// Mitsubishi GX Works2 project: DGPTapM6FX3G   PLC: FX3G

// global labels: Global1
VAR_GLOBAL
  VR1 AT D8030 : INT;
  VR2 AT D8031 : INT;
  XXLimitN AT M8344 : BOOL;
  XXLimitP AT M8343 : BOOL;
  XXBusy AT M8340 : BOOL;
  XXInterruptInverse AT M8347 : BOOL;
  XXPos AT D8340 : DINT;
  XXAccelTime AT D8348 : INT;
  XXDecelTime AT D8349 : INT;
  XXPosView AT D0 : DINT;
  XXTarPos AT D2 : DINT;
  XXFeed AT D4 : DINT;
  XXTarR AT M0 : BOOL;
  XXTarRSkip AT D6 : INT;
  XXOn AT M1 : BOOL;
  XXRun AT M2 : BOOL;
  XXDirection AT M3 : BOOL;
  XXMinI AT X000 : BOOL;
  XXReadyI AT X003 : BOOL;
  XXPulseO AT Y000 : BOOL;
  XXDirectionO AT Y004 : BOOL;
  XXOnO AT Y002 : BOOL;
  YYLimitN AT M8354 : BOOL;
  YYLimitP AT M8353 : BOOL;
  YYBusy AT M8350 : BOOL;
  YYInterruptInverse AT M8357 : BOOL;
  YYPos AT D8350 : DINT;
  YYAccelTime AT D8358 : INT;
  YYDecelTime AT D8359 : INT;
  YYPosView AT D7 : DINT;
  YYTarPos AT D9 : DINT;
  YYFeed AT D11 : DINT;
  YYTarR AT M4 : BOOL;
  YYTarRSkip AT D13 : INT;
  YYOn AT M5 : BOOL;
  YYRun AT M6 : BOOL;
  YYDirection AT M7 : BOOL;
  YYMinI AT X001 : BOOL;
  YYMaxI AT X002 : BOOL;
  YYReadyI AT X004 : BOOL;
  YYPulseO AT Y001 : BOOL;
  YYDirectionO AT Y005 : BOOL;
  YYOnO AT Y003 : BOOL;
  Run AT M8 : BOOL;
  RunI AT X005 : BOOL;
  RunStop AT M9 : BOOL;
  RunStopI AT X006 : BOOL;
  RunState AT D14 : INT;
  RunStateNext AT M10 : BOOL;
  AxisTravelState AT D15 : INT;
  AxisTravelStateNext AT M11 : BOOL;
  AxisTapState AT D16 : INT;
  AxisTapStateNext AT M12 : BOOL;
  FoilState AT D17 : INT;
  FoilStateNext AT M13 : BOOL;
  FoilTopN AT M14 : BOOL;
  FoilTopP AT M15 : BOOL;
  FoilTopPI AT X007 : BOOL;
  FoilTopTimer AT TC0 : BOOL;
  FoilTopTimerDelay AT D18 : INT;
  FoilTop AT M16 : BOOL;
  FoilTopO AT Y006 : BOOL;
  FoilBotN AT M17 : BOOL;
  FoilBotP AT M18 : BOOL;
  FoilBotPI AT X010 : BOOL;
  FoilBotTimer AT TC1 : BOOL;
  FoilBotTimerDelay AT D19 : INT;
  FoilBot AT M19 : BOOL;
  FoilBotO AT Y007 : BOOL;
  OverloadI AT X011 : BOOL;
  WorkFeedTravel AT D20 : DINT;
  WorkFeedTap AT D22 : DINT;
  TravelArray AT D24 : ARRAY [0..1] OF DINT;
  TravelIndex AT D28 : INT;
END_VAR

// task Task_01 (event TRUE, interval 0, priority 31): POU_01

PROGRAM POU_01
VAR
  fTmp : BOOL;
END_VAR
RST(M8002, XXOn);
RST(M8002, YYOn);
MOV(M8002, 100, XXAccelTime);
MOV(M8002, 100, XXDecelTime);
MOV(M8002, 200, YYAccelTime);
MOV(M8002, 200, YYDecelTime);
RST(M8002, FoilTop);
SET(M8002, FoilBot);
(*1000 pulse = 1 mm, 1 round = 2.0mm, -> servo ppr = 2000*)
DMOV(M8002, (2000 * 2850) / 60, WorkFeedTravel);
DMOV(M8002, 5_000, TravelArray[0]);
DMOV(M8002, TravelArray[0] + 42_000, TravelArray[1]);
(*1000 pulse = 1 mm, 1 round = 1.0mm, -> servo ppr = 1000*)
DMOV(M8002, (1000 * 2000) / 60, WorkFeedTap);
(*|||||||||||||||*)
(*|||||||||||||||*)
SET(Run AND RunState = 0, fTmp);
RST(fTmp, Run);
SET(fTmp, XXOn);
MOV(fTmp, 1, RunState);
RST(fTmp, fTmp);
SET(RunStop, fTmp);
RST(fTmp, Run);
RST(fTmp, RunStop);
ZRST(fTmp, RunState, FoilState);
RST(fTmp, XXRun);
RST(fTmp, YYRun);
RST(fTmp, FoilTop);
SET(fTmp, FoilBot);
RST(fTmp, fTmp);
(*|||||||||||||||*)
(*|||||||||||||||*)
INC(RunStateNext, RunState);
INC(AxisTravelStateNext, AxisTravelState);
INC(AxisTapStateNext, AxisTapState);
INC(FoilStateNext, FoilState);
ZRST(M8000, RunStateNext, FoilStateNext);
DECO(M8000, RunState, 6, M100);
DECO(M8000, AxisTravelState, 6, M200); DECO(M8000, AxisTravelState, 6, M1200); ZRST(NOT XXTarR OR NOT XXReadyI, M1200, M1263);
DECO(M8000, AxisTapState, 6, M300); DECO(M8000, AxisTapState, 6, M1300); ZRST(NOT YYTarR OR NOT YYReadyI, M1300, M1363);
DECO(M8000, FoilState, 6, M400);
(*|||||||||||||||*)

(*|||||||||||||||*)
(*origin foil and tap*)
MOV(M101, 1, AxisTapState);
MOV(M101, 1, FoilState);
SET(M101, RunStateNext);
(*origin travel*)
MOV(M102 AND M1320, 1, AxisTravelState);
SET(M102 AND M1320, RunStateNext);
(*ready done, wait run command*)
SET(M103 AND Run, RunStateNext);
(*cycle start*)
SET(M104 AND M1220 AND M1320 AND M420, RunStateNext);
(*travel to hole*)
MOV(M105, 11, AxisTravelState);
SET(M105, RunStateNext);
(*tap*)
MOV(M106 AND M1220, 11, AxisTapState);
SET(M106 AND M1220, RunStateNext);
(*tap done, drop*)
MOV(M105 AND M1320, 11, FoilState);
SET(M105 AND M1320, RunStateNext);
(*drop done, back to cycle start*)
MOV(M106 AND M420, 3, RunState);
(*|||||||||||||||*)

(*|||||||||||||||*)
(*/////get origin travel*)
(*at min, jump to move forward*)
SET(M1201 AND XXMinI, fTmp);
MOV(fTmp, 3, AxisTravelState); RST(fTmp, fTmp);
(*not at min, move back*)
SET(M1201 AND NOT XXMinI, fTmp);
RST(fTmp, XXPos);
DMOV(fTmp, -50_000, XXTarPos);
DMOV(fTmp, 5_000, XXFeed);
SET(fTmp, XXRun);
SET(fTmp, AxisTravelStateNext); RST(fTmp, fTmp);
(*move back hit limit, reset*)
SET(M202 AND NOT XXBusy, fTmp);
RST(fTmp, XXRun);
RST(fTmp, XXPos);
SET(fTmp, AxisTravelStateNext); RST(fTmp, fTmp);
(*move forward*)
SET(M1203, fTmp);
DMOV(fTmp, 5_000, XXTarPos);
DMOV(fTmp, 1_000, XXFeed);
SET(fTmp, XXRun);
SET(fTmp, AxisTravelStateNext); RST(fTmp, fTmp);
(*move forward out min, stop*)
SET(M204 AND NOT XXMinI, fTmp);
RST(fTmp, XXRun);
SET(fTmp, AxisTravelStateNext); RST(fTmp, fTmp);
(*stop done, move forward 1mm*)
SET(M1205, fTmp);
DMOV(fTmp, XXPos + 1000, XXTarPos);
DMOV(fTmp, 1000, XXFeed);
SET(fTmp, XXRun);
SET(fTmp, AxisTravelStateNext); RST(fTmp, fTmp);
(*move forward 1mm done, ready*)
SET(M1206, fTmp);
RST(fTmp, XXPos);
RST(fTmp, TravelIndex);
MOV(fTmp, 20, AxisTravelState); RST(fTmp, fTmp);
(*/////main sequence*)
MOV(M20, (TravelIndex + 1) MOD 2, TravelIndex);
RST(M20, M20);
(*move to hole*)
SET(M1211, fTmp);
DMOV(fTmp, TravelArray[TravelIndex], XXTarPos);
DMOV(fTmp, WorkFeedTap, XXFeed);
MOV(fTmp, (TravelIndex + 1) MOD 2, TravelIndex);
SET(fTmp, XXRun);
SET(fTmp, AxisTravelStateNext); RST(fTmp, fTmp);
(*target reach or touch max, reset*)
SET(M1212 OR (M212 AND NOT XXBusy), fTmp);
RST(fTmp, XXRun);
SET(fTmp, AxisTravelStateNext); RST(fTmp, fTmp);
(*move to hole done, end*)
SET(M1213, fTmp);
MOV(fTmp, 20, AxisTravelState); RST(fTmp, fTmp);
(*|||||||||||||||*)


(*|||||||||||||||*)
(*/////get origin tap*)
(*at min, jump to move down*)
SET(M1301 AND YYMinI, fTmp);
MOV(fTmp, 3, AxisTapState); RST(fTmp, fTmp);
(*not at min, move up*)
SET(M1301 AND NOT YYMinI, fTmp);
RST(fTmp, YYPos);
DMOV(fTmp, -50_000, YYTarPos);
DMOV(fTmp, 5_000, YYFeed);
SET(fTmp, YYRun);
SET(fTmp, AxisTapStateNext); RST(fTmp, fTmp);
(*move up hit limit, reset*)
SET(M302 AND NOT YYBusy, fTmp);
RST(fTmp, YYRun);
RST(fTmp, YYPos);
SET(fTmp, AxisTapStateNext); RST(fTmp, fTmp);
(*move down*)
SET(M1303, fTmp);
DMOV(fTmp, 5_000, YYTarPos);
DMOV(fTmp, 1_000, YYFeed);
SET(fTmp, YYRun);
SET(fTmp, AxisTapStateNext); RST(fTmp, fTmp);
(*move down out min, stop*)
SET(M304 AND NOT YYMinI, fTmp);
RST(fTmp, YYRun);
SET(fTmp, AxisTapStateNext); RST(fTmp, fTmp);
(*stop done, move down 1mm*)
SET(M1305, fTmp);
DMOV(fTmp, YYPos + 1000, YYTarPos);
DMOV(fTmp, 1000, YYFeed);
SET(fTmp, YYRun);
SET(fTmp, AxisTapStateNext); RST(fTmp, fTmp);
(*move down 1mm done, ready*)
SET(M1306, fTmp);
RST(fTmp, YYPos);
MOV(fTmp, 20, AxisTapState); RST(fTmp, fTmp);
(*/////main sequence*)
(*wait run hit, move down*)
SET(M1311, fTmp);
DMOV(fTmp, 32_000, YYTarPos);
DMOV(fTmp, WorkFeedTap, YYFeed);
SET(fTmp, YYRun);
SET(fTmp, AxisTapStateNext); RST(fTmp, fTmp);
(*target reach or touch max, reset*)
SET(M1312 OR (M312 AND NOT YYBusy), fTmp);
RST(fTmp, YYRun);
SET(fTmp, AxisTapStateNext); RST(fTmp, fTmp);
(*move down slow done, move up*)
SET(M1313, fTmp);
DMOV(fTmp, 0, YYTarPos);
DMOV(fTmp, WorkFeedTap, YYFeed);
SET(fTmp, YYRun);
SET(fTmp, AxisTapStateNext); RST(fTmp, fTmp);
(*move up done, return wait tap hit*)
SET(M1314, fTmp);
MOV(fTmp, 20, AxisTapState); RST(fTmp, fTmp);
(*|||||||||||||||*)

(*|||||||||||||||*)
MOV(M8000, 1 + (VR1 / 16), FoilTopTimerDelay);
MOV(M8000, 1 + (VR2 / 16), FoilBotTimerDelay);
(*get origin*)
SET(M301, FoilTop);
SET(M301, FoilBot);
SET(M301 AND FoilTopP AND FoilBotP, FoilStateNext);
(*get origin done*)
MOV(M302, 20, FoilState);
(*/////main sequence*)
(*bot back, done, next*)
RST(M311, FoilBot);
SET(M311 AND FoilBotN, FoilStateNext);
(*wait drop, bot forward, done, next*)
OUT_T(M312, FoilBotTimer, FoilBotTimerDelay);
SET(FoilBotTimer, FoilBot);
SET(FoilBotTimer AND FoilBotP, FoilStateNext);
(*top back, done, next*)
RST(M313, FoilTop);
SET(M313 AND FoilTopN, FoilStateNext);
(*wait drop, top forward, done, next*)
OUT_T(M314, FoilTopTimer, FoilTopTimerDelay);
SET(FoilTopTimer, FoilTop);
SET(FoilTopTimer AND FoilTopP, FoilStateNext);
(*end*)
MOV(M315, 20, FoilState);
(*|||||||||||||||*)

(*|||||||||||||||*)
(*XX*)
RST(XXRun AND XXTarPos = XXPos, XXRun);
DDRVA(XXRun, XXTarPos, XXFeed, XXPulseO, XXDirection);
RST(M8029, XXRun);
OUT(XXDirection, XXDirectionO);
INC(NOT XXRun AND NOT XXBusy AND XXTarRSkip < 5, XXTarRSkip);
RST(XXRun, XXTarRSkip);
OUT(XXTarRSkip >= 5, XXTarR);
(**)
OUT(XXMinI, XXLimitN);
(*|||||||||||||||*)
(*YY*)
RST(YYRun AND YYTarPos = YYPos, YYRun);
DDRVA(YYRun, YYTarPos, YYFeed, YYPulseO, YYDirection);
RST(M8029, YYRun);
OUT(YYDirection, YYDirectionO);
INC(NOT YYRun AND NOT YYBusy AND YYTarRSkip < 5, YYTarRSkip);
RST(YYRun, YYTarRSkip);
OUT(YYTarRSkip >= 5, YYTarR);
(**)
OUT(YYMinI, YYLimitN);
OUT(YYMaxI, YYLimitP);
(*|||||||||||||||*)

MOV(M8000, 1 + (VR1 / 16), FoilTopTimerDelay);
MOV(M8000, 1 + (VR2 / 16), FoilBotTimerDelay);
(*|||||||||||||||*)
PLS(RunI, Run); SET(Run, Run);
PLS(RunStopI, RunStop); SET(RunStop, RunStop);
PLS(OverloadI, RunStop); SET(RunStop, RunStop);
OUT_T(NOT FoilTop, FoilTopTimer, FoilTopTimerDelay); SET(FoilTopTimer, FoilTopN); RST(FoilTopTimer, FoilTopP);
SET(FoilTopPI, FoilTopP); RST(FoilTopPI, FoilTopN);
OUT_T(NOT FoilBot, FoilBotTimer, FoilBotTimerDelay); SET(FoilBotTimer, FoilBotN); RST(FoilBotTimer, FoilBotP);
SET(FoilBotPI, FoilBotP); RST(FoilBotPI, FoilBotN);
(*|||||||||||||||*)
OUT(XXOn, XXOnO);
OUT(FoilTop, FoilTopO);
OUT(NOT FoilBot, FoilBotO);
(*|||||||||||||||*)
END_PROGRAM
